TYPE Terminal_Input_typ : 	
	STRUCT 
		Par : Terminal_Parameter_typ;
	END_STRUCT
END_TYPE

(* stored: Version 1.1.0.1, ProductVersion 3.1.4024.3
   DUT Terminal_Input_typ: Id {a98c3eb7-d1f0-003e-3afa-5c8166517e6a} *)
